// TIA Portal V18 export
FUNCTION "Analog_Handling" : Void   // FC3, FBD
TITLE = Analog Handling
{ S7_Optimized_Access := 'TRUE' }
VERSION : 0.1
// stored: AutoNumber true, IsIECCheckEnabled false, SetENOAutomatically false, UDAEnableTagReadback false
   VAR_TEMP
      Dummy11 : Bool;
      Dummy21 : Bool;
   END_VAR
BEGIN

REGION Network 1: **************INPUTS*************
END_REGION

REGION Network 2 (SCL): SCL Network
   IF #Dummy1 THEN
       #Dummy2 := FALSE;    // Statement section IF

   END_IF;
END_REGION

REGION Network 3: CI Proportional Valve Input
   // Rexroth Bef Prop Valve
   // IN: 0-27648
   // UT: 0-100
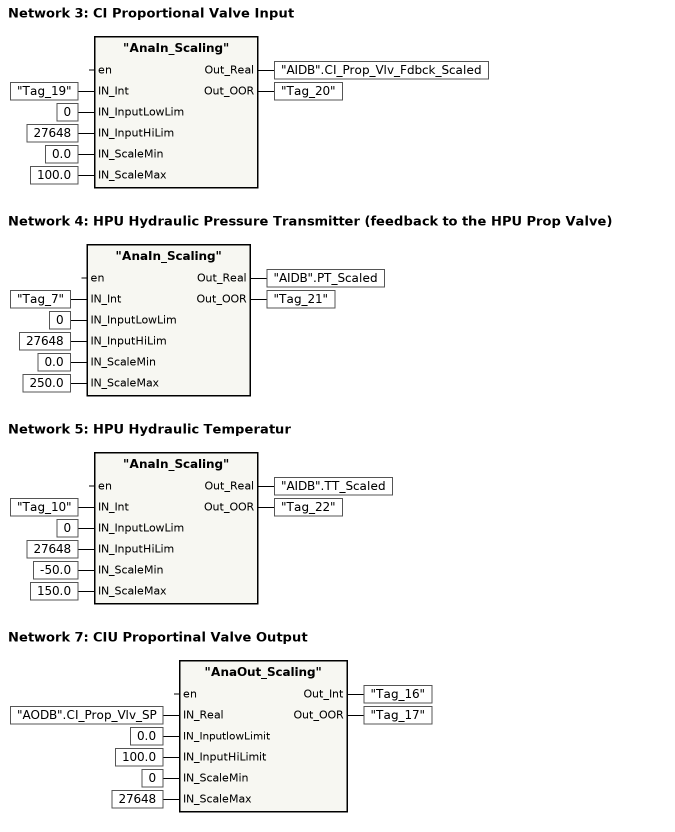
   "AnaIn_Scaling"(IN_Int := "Tag_19",
                   IN_InputLowLim := 0,
                   IN_InputHiLim := 27648,
                   IN_ScaleMin := 0.0,
                   IN_ScaleMax := 100.0,
                   Out_Real => "AIDB".CI_Prop_Vlv_Fdbck_Scaled,
                   Out_OOR => "Tag_20");
END_REGION

REGION Network 4: HPU Hydraulic Pressure Transmitter (feedback to the HPU Prop Valve)
   // IFM PT5401
   // 0-250 bar/4-20mA
   "AnaIn_Scaling"(IN_Int := "Tag_7",
                   IN_InputLowLim := 0,
                   IN_InputHiLim := 27648,
                   IN_ScaleMin := 0.0,
                   IN_ScaleMax := 250.0,
                   Out_Real => "AIDB".PT_Scaled,
                   Out_OOR => "Tag_21");
END_REGION

REGION Network 5: HPU Hydraulic Temperatur
   // IFM TN2435
   // -50...150 grader /4-20mA
   "AnaIn_Scaling"(IN_Int := "Tag_10",
                   IN_InputLowLim := 0,
                   IN_InputHiLim := 27648,
                   IN_ScaleMin := -50.0,
                   IN_ScaleMax := 150.0,
                   Out_Real => "AIDB".TT_Scaled,
                   Out_OOR => "Tag_22");
END_REGION

REGION Network 6: **************OUTPUTS**************
END_REGION

REGION Network 7: CIU Proportinal Valve Output
   "AnaOut_Scaling"(IN_Real := "AODB".CI_Prop_Vlv_SP,
                    IN_InputlowLimit := 0.0,
                    IN_InputHiLimit := 100.0,
                    IN_ScaleMin := 0,
                    IN_ScaleMax := 27648,
                    Out_Int => "Tag_16",
                    Out_OOR => "Tag_17");
END_REGION
END_FUNCTION
